FUNCTION CheckDivReal : REAL
VAR_INPUT
    divisor : REAL;
END_VAR

IF divisor = 0 THEN
    CheckDivReal := 2;
nTooHigh := nTooHigh + 1;
ELSE
    CheckDivReal := divisor;
END_IF

END_FUNCTION

(* stored: Version 1.1.0.1, ProductVersion 3.1.4024.15
   POU CheckDivReal: Id {ad82391b-7d7f-4b56-b937-bf5ae08821ff}, SpecialFunc CheckDivReal32 *)
